(* CODESYS project ControlDeposito.project
   Title: ControlDeposito
   Version: 0.0.0.0
   Author: serbogr1

Project tree, tasks and I/O mapping:
  MyController : TM241CE40R, Schneider Electric, order no. TM241CE40R, version 4.0.6.18
    application Application
      libraries: Toolbox, 2.2.0.0 (Schneider Electric); Util, 3.5.1.0 (System)
      task MAST (cyclic, interval 50 ms, priority 15, watchdog 100 ms x 1) calls Control_PID
      global variables GVL
      program Control_PID [LD]
      visualisation ControlNivel
    DI : Digital Inputs, Schneider Electric, version 4.0.6.18
        input  idwDI_IDW0 : DWORD  // IDW0
        input  ibDI_IB1 : BYTE  // IB1
    DQ : Digital Outputs, Schneider Electric, version 4.0.6.18
        output qwDQ_QW0 : WORD  // QW0
        output qbDQ_QB1 : BYTE  // QB1
    Counters : Counters, Schneider Electric, version 4.0.6.18
    Pulse_Generators : Pulse Generators, Schneider Electric, version 4.0.6.18
    Cartridge_1 : Cartridge, Schneider Electric, version 4.0.6.18
    Cartridge_2 : Cartridge, Schneider Electric, version 4.0.6.18
    IO_Bus : IO bus - TM3, Schneider Electric, version 4.0.6.18
    COM_Bus : COM bus, Schneider Electric, version 4.0.6.18
    Ethernet_1 : Ethernet Network, Schneider Electric, version 4.0.6.18
        settings: IPAddress = [172, 16, 191, 108]; SubnetMask = [255, 255, 255, 0]; GatewayAddress = [172, 16, 191, 1]; WebServer = TRUE; FTP Server = TRUE; SoMachine Protocol = TRUE; Modbus Server = TRUE; NetManage Protocol = TRUE; SNMP protocol = TRUE; Enable Routing = FALSE; WebVisu protocol = TRUE; DHCP Server Active = FALSE
    Serial_Line_1 : Serial line, Schneider Electric, version 4.0.6.18
      SoMachine_Network_Manager : SoMachine-Network Manager, Schneider Electric, version 4.0.0.2
    Serial_Line_2 : Serial line, Schneider Electric, version 4.0.6.18
      Modbus_Manager : Modbus Manager, Schneider Electric, version 4.0.0.2
  text list GlobalTextList
*)

// MyController/Application/GVL
VAR_GLOBAL
END_VAR

// MyController/Application/Control_PID
PROGRAM Control_PID
VAR
	tru: BOOL;
	Escalado_Nivel: FB_Scaling;
	PID_ControNivel: Util.PID;
	Escalado_valvula_Descarga: SE_TBX.FB_Scaling;
	AutoManual: BOOL;
	ResetPID: BOOL;
END_VAR
VAR
	wNivel AT %MW1: WORD;
	wFlujo AT %MW0: WORD;
	wValvulaLlenado AT %MW2: WORD := 500;
	wValvulaDescarga AT %MW3: WORD;
	bLuzStart AT %QX0.0: BOOL;
	bLuzStop AT %QX0.1: BOOL;
	bLuzReset AT %QX0.2: BOOL;
	rNivel: REAL;
	rFlujo: REAL;
	rValvulaLlenado: REAL;
	rValvulaDescarga: REAL;
	rReferencia: REAL;
END_VAR

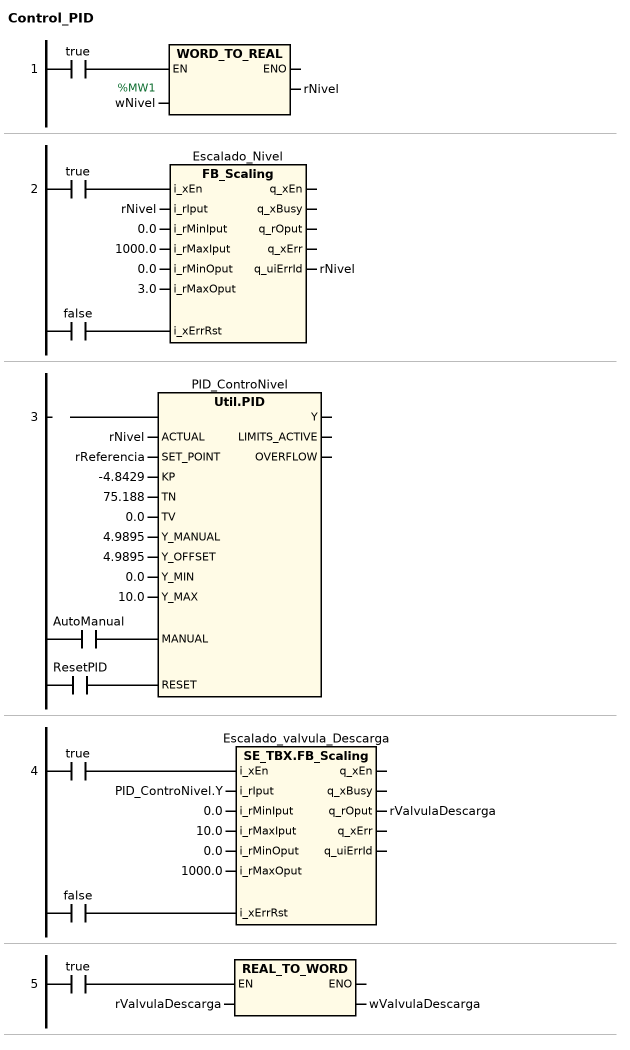
// NETWORK 1
//   wNivel: AT %MW1
IF true THEN rNivel := WORD_TO_REAL(wNivel); END_IF

// NETWORK 2
Escalado_Nivel(
    i_xEn := true,
    i_rIput := rNivel,
    i_rMinIput := 0.0,
    i_rMaxIput := 1000.0,
    i_rMinOput := 0.0,
    i_rMaxOput := 3.0,
    i_xErrRst := false,
    q_uiErrId => rNivel); // FB_Scaling

// NETWORK 3
PID_ControNivel(
    ACTUAL := rNivel,
    SET_POINT := rReferencia,
    KP := -4.8429,
    TN := 75.188,
    TV := 0.0,
    Y_MANUAL := 4.9895,
    Y_OFFSET := 4.9895,
    Y_MIN := 0.0,
    Y_MAX := 10.0,
    MANUAL := AutoManual,
    RESET := ResetPID); // Util.PID

// NETWORK 4
//   PID_ControNivel.Y: manipulated variable, set value
Escalado_valvula_Descarga(
    i_xEn := true,
    i_rIput := PID_ControNivel.Y,
    i_rMinIput := 0.0,
    i_rMaxIput := 10.0,
    i_rMinOput := 0.0,
    i_rMaxOput := 1000.0,
    i_xErrRst := false,
    q_rOput => rValvulaDescarga); // SE_TBX.FB_Scaling

// NETWORK 5
//   wValvulaDescarga: AT %MW3
IF true THEN wValvulaDescarga := REAL_TO_WORD(rValvulaDescarga); END_IF

END_PROGRAM

// MyController/Application/ControlNivel
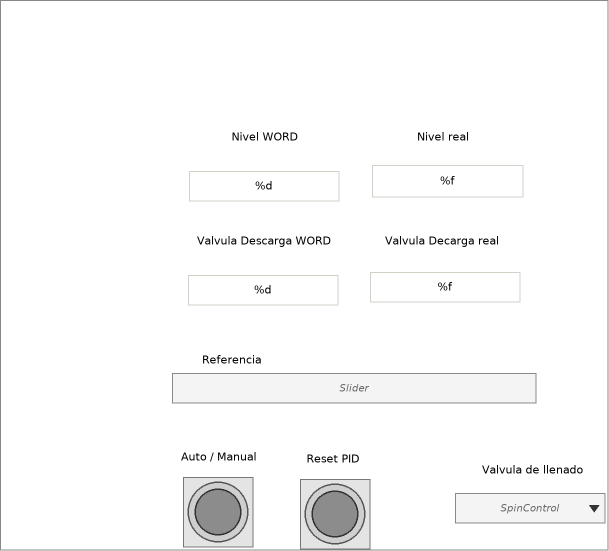
VISUALIZATION ControlNivel  // 609x551
    Textfield (189,171 150x30), "%d", text variable: Control_PID.wNivel
    Textfield (372,165 151x32), "%f", text variable: Control_PID.rNivel
    Label (190,122 150x30), "Nivel WORD"
    Label (368,122 150x30), "Nivel real"
    Textfield (188,275 150x30), "%d", text variable: Control_PID.wFlujo
    Textfield (370,272 150x30), "%f", text variable: Control_PID.rValvulaDescarga
    Label (189,226 150x30), "Valvula Descarga WORD"
    Label (367,226 150x30), "Valvula Decarga real"
    Slider (172,373 364x30), variable: Control_PID.rReferencia, scale 0..3
    Label (157,345 150x30), "Referencia"
    PushSwitchLed (183,477 70x70), variable: Control_PID.AutoManual, behaviour: TOGGLE, style: Switch-PushSwitchLed-Gray
    Label (144,442 150x30), "Auto / Manual"
    PushSwitchLed (300,479 70x70), variable: Control_PID.ResetPID, behaviour: TOGGLE, style: Switch-PushSwitchLed-Gray
    Label (258,444 150x30), "Reset PID"
    SpinControl (455,493 150x30), variable: Control_PID.wValvulaLlenado
    Label (458,455 149x30), "Valvula de llenado"
END_VISUALIZATION
